# EPICS StreamDevice protocol: protocols/intmon.proto
Terminator = LF;
ExtraInput = Ignore;

trig {
# fin kHz, fout (setpoint)
	out "y";
	in;
}

irq {
	in "\$1 %d %*s";
}

irqs {
	in "\$1 %*d %s";
}
